(* Logix 5000 project; controller StartingFile_Isaiah_Regacho vendor 1 type 14 code 106 rev 28.11; software revision 28.03; part 2 of 2 *)
(* tags used below, declared in another part *)
   callArray : DINT[6];
   clearFaultsBit : BOOL;
   Current_State : DINT;
   currentFloor : DINT;
   doorOpenFault : TIMER;
   doorOpenFault_ons : BOOL;
   doorOpenFaultBit : BOOL;
   elevatorDirection : DINT;
   floor1 : DINT;
   floor1_ons : BOOL;
   floor1Data : getFloorData;
   floor2 : DINT;
   floor2_ons : BOOL;
   floor2Data : getFloorData;
   floor3 : DINT;
   floor3_ons : BOOL;
   floor3Data : getFloorData;
   floor4 : DINT;
   floor4_ons : BOOL;
   floor4Data : getFloorData;
   index : DINT;
   majorFault_var : DINT;
   masterFaultLog : FAULTS[10];
   masterLogData : LOG_DATA[4];
   motorRunFault : TIMER;
   motorRunFault_ons : BOOL;
   motorRunFaultBit : BOOL;
   Next_State : DINT;
   nextFloor : DINT;
   sensorFault_ons : BOOL;
   sensorFaultBit : BOOL;
   START : ALIAS FOR Local:2:I.Data.14;   // Start Button (N.O.)
   V_CR0 : BOOL;   // Virtual Control Relay 0
   V_DCLS : BOOL;   // Virtual Door Close Limit Switch
   V_FIL1 : BOOL;   // Virtual Floor Indicator Light 1
   V_FIL2 : BOOL;   // Virtual Floor Indicator Light 2
   V_FIL3 : BOOL;   // Virtual Floor Indicator Light 3
   V_FIL4 : BOOL;   // Virtual Floor Indicator Light 4
   V_FLS1 : BOOL;   // Virtual Floor Limit Switch 1
   V_FLS2 : BOOL;   // Virtual Floor Limit Switch 2
   V_FLS3 : BOOL;   // Virtual Floor Limit Switch 3
   V_FLS4 : BOOL;   // Virtual Floor Limit Switch 4
   V_FPB1 : BOOL;   // Virtual Floor Pushbutton 1
   V_FPB2 : BOOL;   // Virtual Floor Pushbutton 2
   V_FPB3 : BOOL;   // Virtual Floor Pushbutton 3
   V_FPB4 : BOOL;   // Virtual Floor Pushbutton 4
   V_IL1 : BOOL;   // Virtual Indicator Light 1
   V_IL2 : BOOL;   // Virtual Indicator Light 2
   V_IL3 : BOOL;   // Virtual Indicator Light 3
   V_IL4 : BOOL;   // Virtual Indicator Light 4
   V_ILE5 : BOOL;   // Virtual Indicator Light Emergency 5
   V_M0 : BOOL;   // Virtual Motor 0
   V_PB1 : BOOL;   // Virtual Pushbutton 1
   V_PB2 : BOOL;   // Virtual Pushbutton 2
   V_PB3 : BOOL;   // Virtual Pushbutton 3
   V_PB4 : BOOL;   // Virtual Pushbutton 4
   V_SOL0 : BOOL;   // Virtual Solenoid 0
   V_START : BOOL;   // Virtual Start Button (N.O.)
(* MainProgram, continued *)

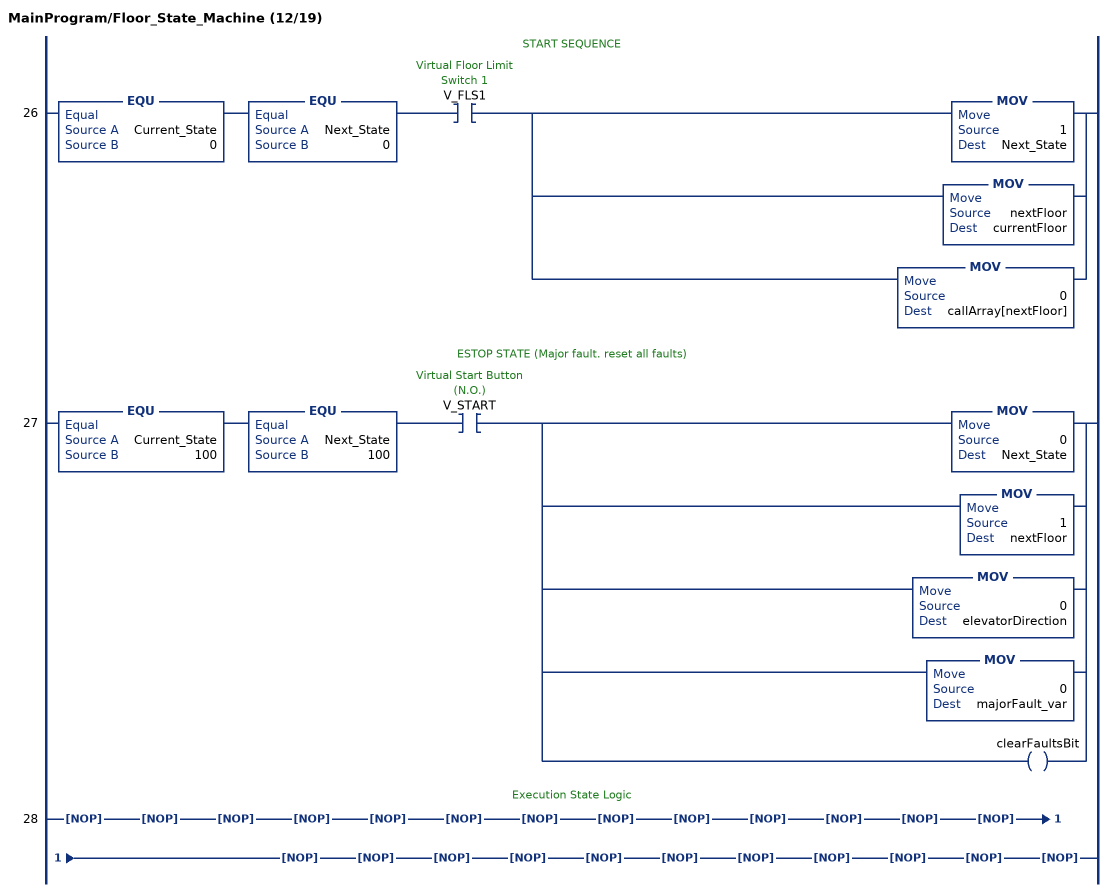
   // START SEQUENCE
   26: EQU(Current_State,0)EQU(Next_State,0)XIC(V_FLS1)[MOV(1,Next_State) ,MOV(nextFloor,currentFloor) ,MOV(0,callArray[nextFloor]) ];
   // ESTOP STATE (Major fault. reset all faults)
   27: EQU(Current_State,100)EQU(Next_State,100)XIC(V_START)[MOV(0,Next_State) ,MOV(1,nextFloor) ,MOV(0,elevatorDirection) ,MOV(0,majorFault_var) ,OTE(clearFaultsBit) ];
   // Execution State Logic
   28: NOP()NOP()NOP()NOP()NOP()NOP()NOP()NOP()NOP()NOP()NOP()NOP()NOP()NOP()NOP()NOP()NOP()NOP()NOP()NOP()NOP()NOP()NOP()NOP();
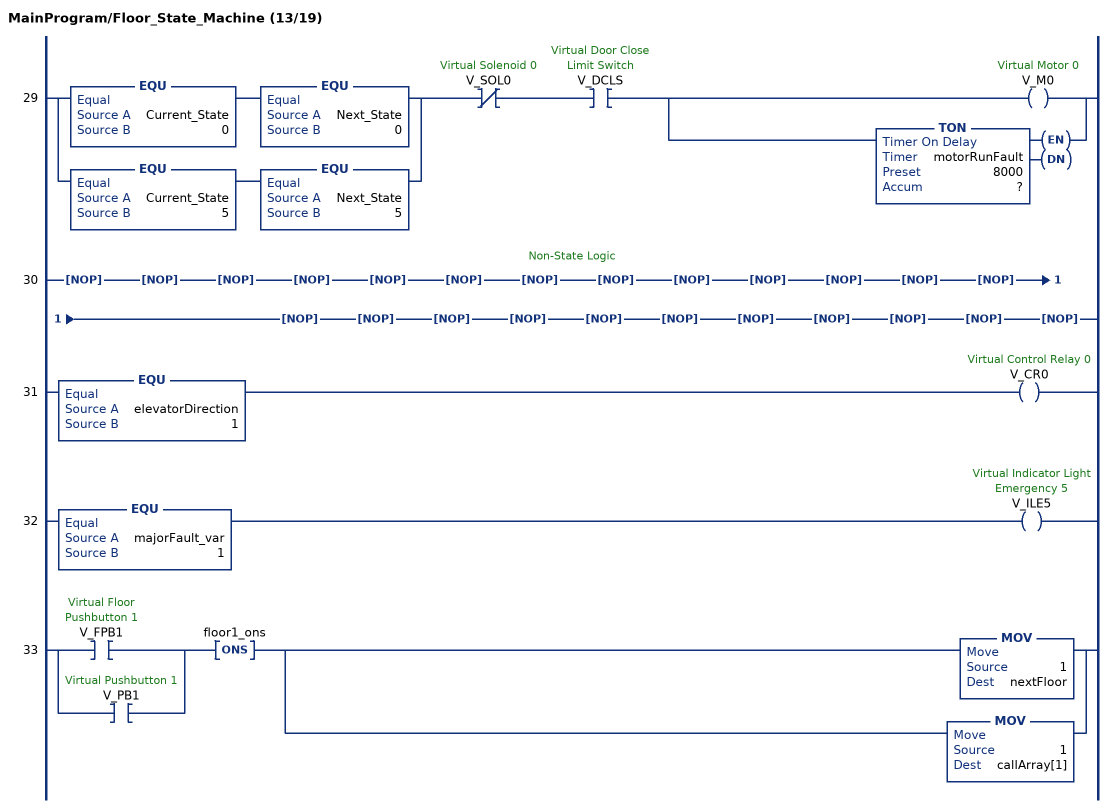
   29: [EQU(Current_State,0) EQU(Next_State,0) ,EQU(Current_State,5) EQU(Next_State,5) ]XIO(V_SOL0)XIC(V_DCLS)[OTE(V_M0) ,TON(motorRunFault,?,?) ];
   // Non-State Logic
   30: NOP()NOP()NOP()NOP()NOP()NOP()NOP()NOP()NOP()NOP()NOP()NOP()NOP()NOP()NOP()NOP()NOP()NOP()NOP()NOP()NOP()NOP()NOP()NOP();
   31: EQU(elevatorDirection,1)OTE(V_CR0);
   32: EQU(majorFault_var,1)OTE(V_ILE5);
   33: [XIC(V_FPB1) ,XIC(V_PB1) ]ONS(floor1_ons)[MOV(1,nextFloor) ,MOV(1,callArray[1]) ];
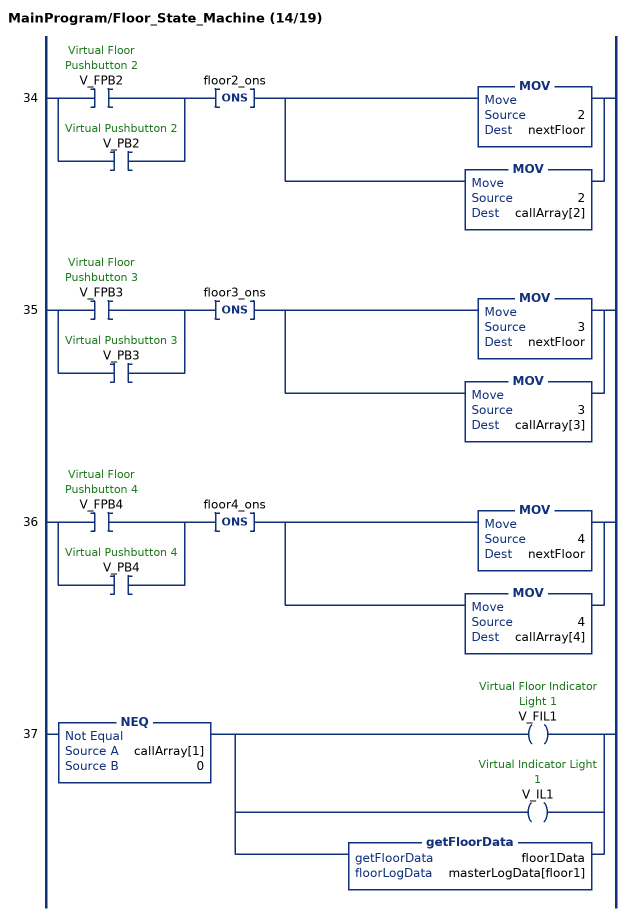
   34: [XIC(V_FPB2) ,XIC(V_PB2) ]ONS(floor2_ons)[MOV(2,nextFloor) ,MOV(2,callArray[2]) ];
   35: [XIC(V_FPB3) ,XIC(V_PB3) ]ONS(floor3_ons)[MOV(3,nextFloor) ,MOV(3,callArray[3]) ];
   36: [XIC(V_FPB4) ,XIC(V_PB4) ]ONS(floor4_ons)[MOV(4,nextFloor) ,MOV(4,callArray[4]) ];
   37: NEQ(callArray[1],0)[OTE(V_FIL1) ,OTE(V_IL1) ,getFloorData(floor1Data,masterLogData[floor1]) ];
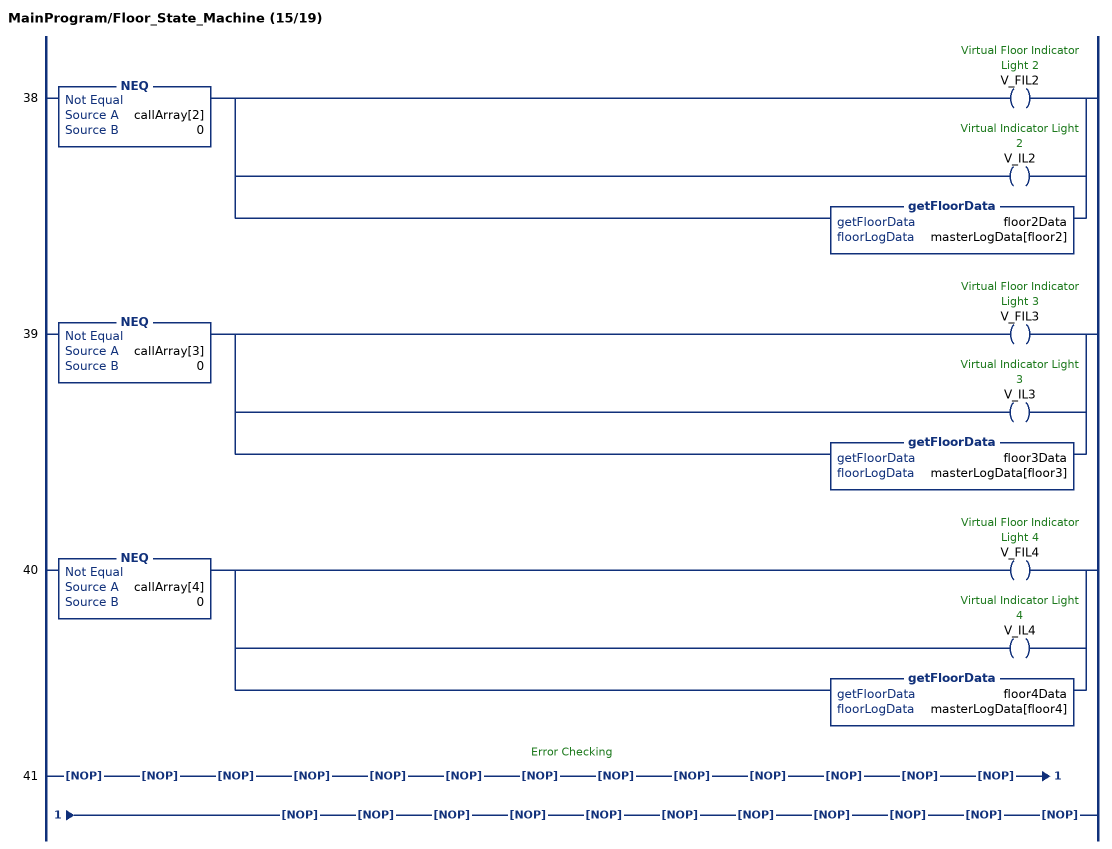
   38: NEQ(callArray[2],0)[OTE(V_FIL2) ,OTE(V_IL2) ,getFloorData(floor2Data,masterLogData[floor2]) ];
   39: NEQ(callArray[3],0)[OTE(V_FIL3) ,OTE(V_IL3) ,getFloorData(floor3Data,masterLogData[floor3]) ];
   40: NEQ(callArray[4],0)[OTE(V_FIL4) ,OTE(V_IL4) ,getFloorData(floor4Data,masterLogData[floor4]) ];
   // Error Checking
   41: NOP()NOP()NOP()NOP()NOP()NOP()NOP()NOP()NOP()NOP()NOP()NOP()NOP()NOP()NOP()NOP()NOP()NOP()NOP()NOP()NOP()NOP()NOP()NOP();
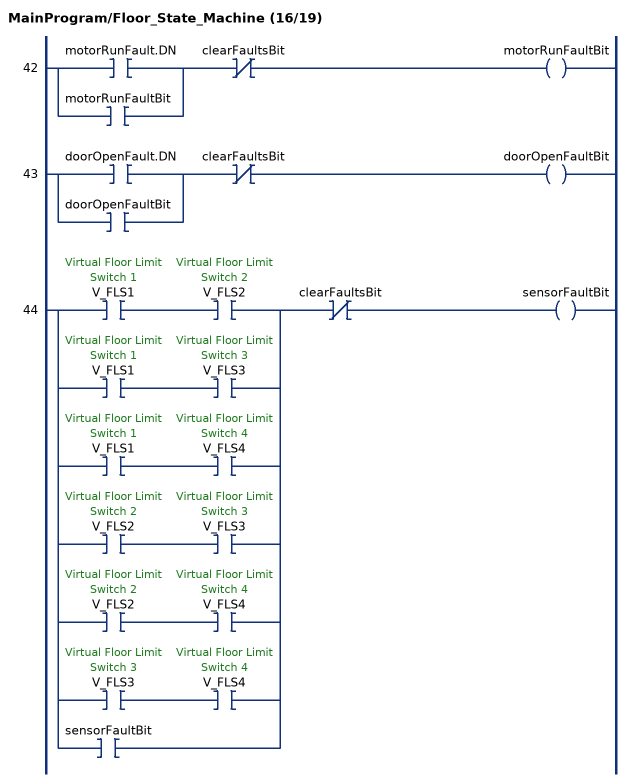
   42: [XIC(motorRunFault.DN) ,XIC(motorRunFaultBit) ]XIO(clearFaultsBit)OTE(motorRunFaultBit);
   43: [XIC(doorOpenFault.DN) ,XIC(doorOpenFaultBit) ]XIO(clearFaultsBit)OTE(doorOpenFaultBit);
   44: [XIC(V_FLS1) XIC(V_FLS2) ,XIC(V_FLS1) XIC(V_FLS3) ,XIC(V_FLS1) XIC(V_FLS4) ,XIC(V_FLS2) XIC(V_FLS3) ,XIC(V_FLS2) XIC(V_FLS4) ,XIC(V_FLS3) XIC(V_FLS4) ,XIC(sensorFaultBit) ]XIO(clearFaultsBit)OTE(sensorFaultBit);
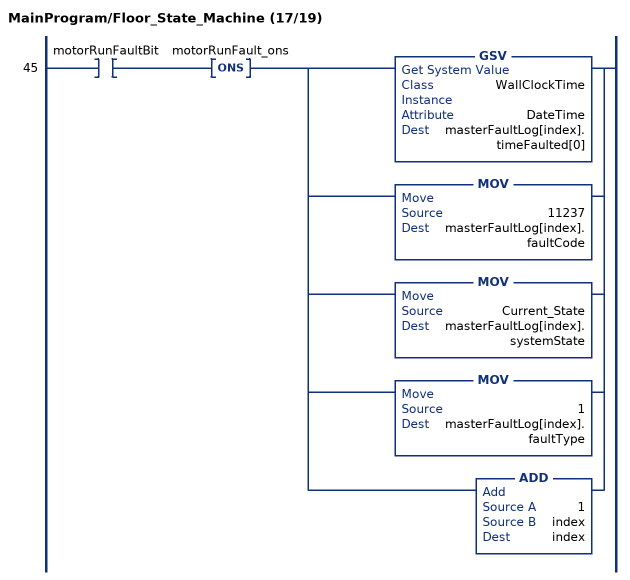
   45: XIC(motorRunFaultBit)ONS(motorRunFault_ons)[GSV(WallClockTime,,DateTime,masterFaultLog[index].timeFaulted[0]) ,MOV(11237,masterFaultLog[index].faultCode) ,MOV(Current_State,masterFaultLog[index].systemState) ,MOV(1,masterFaultLog[index].faultType) ,ADD(1,index,index) ];
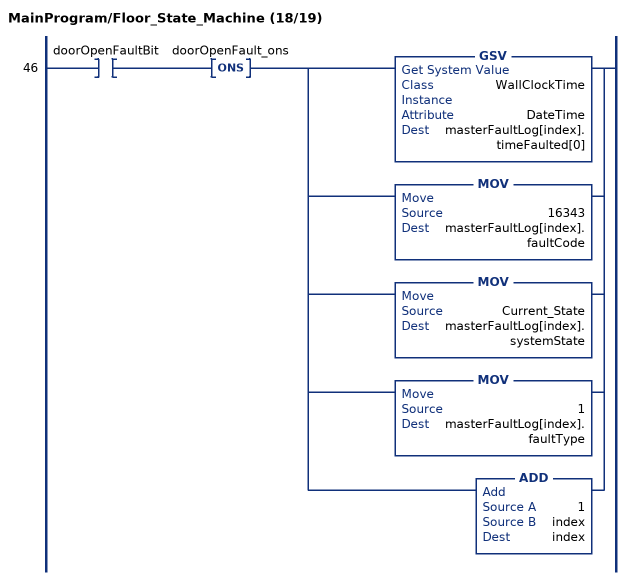
   46: XIC(doorOpenFaultBit)ONS(doorOpenFault_ons)[GSV(WallClockTime,,DateTime,masterFaultLog[index].timeFaulted[0]) ,MOV(16343,masterFaultLog[index].faultCode) ,MOV(Current_State,masterFaultLog[index].systemState) ,MOV(1,masterFaultLog[index].faultType) ,ADD(1,index,index) ];
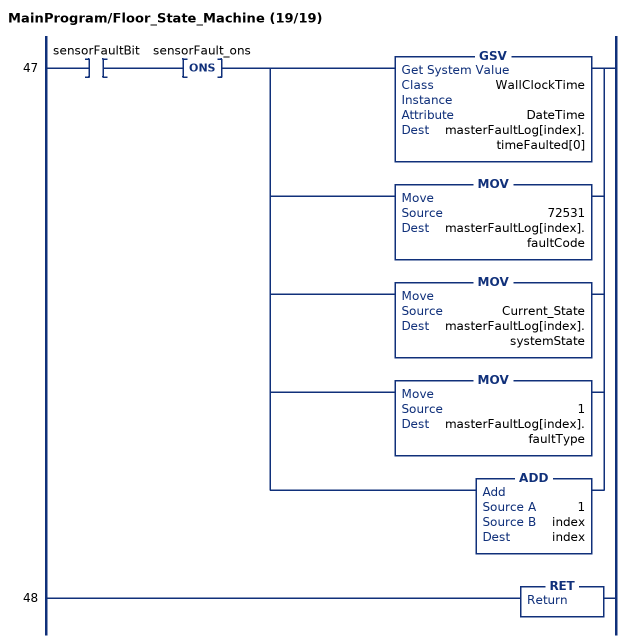
   47: XIC(sensorFaultBit)ONS(sensorFault_ons)[GSV(WallClockTime,,DateTime,masterFaultLog[index].timeFaulted[0]) ,MOV(72531,masterFaultLog[index].faultCode) ,MOV(Current_State,masterFaultLog[index].systemState) ,MOV(1,masterFaultLog[index].faultType) ,ADD(1,index,index) ];
   48: RET();
END_ROUTINE

ROUTINE MainRoutine   (* ladder *)
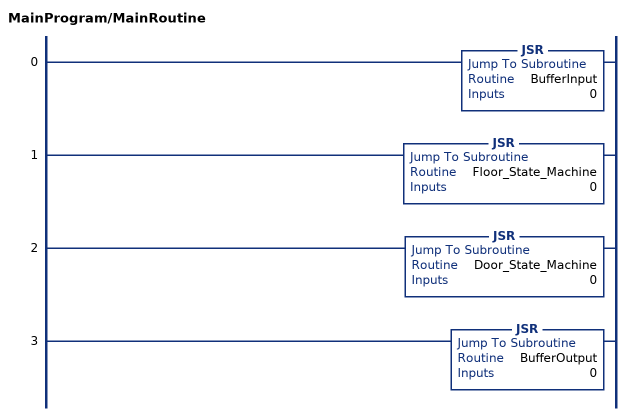
   0: JSR(BufferInput,0);
   1: JSR(Floor_State_Machine,0);
   2: JSR(Door_State_Machine,0);
   3: JSR(BufferOutput,0);
END_ROUTINE
END_PROGRAM
